TYPE ST_DigitalInputParCfg :
STRUCT
    SchemaVersion : UINT := 1; // §3.8: first member even when the passive type has no behavior parameter
END_STRUCT
END_TYPE

(* stored: Version 1.1.0.1, ProductVersion 3.1.4024.12
   DUT ST_DigitalInputParCfg: Id {f543db6b-e72f-4836-948c-3a931f60643d} *)
